FUNCTION_BLOCK JsonGraphSettingsParser IMPLEMENTS I_GraphSettings
VAR
	parser : FB_JsonDomParser;
	baseJsonValue : SJsonValue;
	jsonLanguagePack : I_JsonLanguagePack;

	_nodeCount : UDINT;
	_lastNodeId : NodeId;
	_lastLinkId : T_MAXSTRING;
	
	nodeParser : JsonNodeSettingsParser(0);
	linkParser : JsonLinkSettingsParser(0);
END_VAR

METHOD PUBLIC Clear
VAR_INPUT
END_VAR
baseJsonValue := 0;
parser.NewDocument();
END_METHOD

METHOD FB_init : BOOL
VAR_INPUT
	bInitRetains : BOOL; // if TRUE, the retain variables are initialized (warm start / cold start)
	bInCopyCode : BOOL;  // if TRUE, the instance afterwards gets moved into the copy code (online change)
	JsonLanguagePack : I_JsonLanguagePack;
END_VAR
THIS^.jsonLanguagePack := JsonLanguagePack;

nodeParser.FB_init(bInitRetains, bInCopyCode, JsonLanguagePack);
linkParser.FB_init(bInitRetains, bInCopyCode, JsonLanguagePack);
END_METHOD

METHOD PUBLIC GetLinkById : I_LinkSettings
VAR_INPUT
	Id : T_MAXSTRING;
END_VAR
VAR
	i: UDINT;
END_VAR
FOR i := 0 TO LinkCount - 1  DO
	
	linkParser.Update(parser,GetLinkObjectByIndex(i));
	
	IF linkParser.Id = Id THEN
		GetLinkById := linkParser;
		return;
	END_IF

END_FOR
END_METHOD

METHOD PUBLIC GetLinkByIndex : I_LinkSettings
VAR_INPUT
	Index : UDINT;
END_VAR
linkParser.Update(parser,GetLinkObjectByIndex(Index));
GetLinkByIndex := linkParser;
END_METHOD

METHOD PRIVATE GetLinkObjectByIndex : SJsonValue
VAR_INPUT
	Index : UDINT;
END_VAR
GetLinkObjectByIndex := parser.GetArrayValueByIdx(GetLinksArray(), Index);
END_METHOD

METHOD PRIVATE GetLinksArray : SJsonValue
GetLinksArray := parser.FindMember(baseJsonValue, 'links');
END_METHOD

METHOD PUBLIC GetNodeById : I_NodeSettings
VAR_INPUT
	Id : NodeId;
END_VAR
VAR
	i: UDINT;
END_VAR
FOR i := 0 TO NodeCount - 1  DO
	
	nodeParser.Update(parser,GetNodeObjectByIndex(i));
	
	IF nodeParser.Id = Id THEN
		GetNodeById := nodeParser;
		return;
	END_IF

END_FOR
END_METHOD

METHOD PUBLIC GetNodeByIndex : I_NodeSettings
VAR_INPUT
	Index : UDINT;
END_VAR
nodeParser.Update(parser,GetNodeObjectByIndex(Index));
GetNodeByIndex := nodeParser;
END_METHOD

METHOD PRIVATE GetNodeObjectByIndex : SJsonValue
VAR_INPUT
	Index : UDINT;
END_VAR
GetNodeObjectByIndex := parser.GetArrayValueByIdx(GetNodesArray(),Index);
END_METHOD

METHOD PRIVATE GetNodesArray : SJsonValue
GetNodesArray := parser.FindMember(baseJsonValue, 'nodes');
END_METHOD

PROPERTY PUBLIC HasLinks : Bool
GET
VAR
	tempJsonValue: SJsonValue;
END_VAR
tempJsonValue := GetLinksArray();

IF tempJsonValue = 0 OR_ELSE NOT parser.IsArray(tempJsonValue) THEN
	RETURN;	
END_IF

HasLinks := TRUE;
END_GET
END_PROPERTY

PROPERTY PUBLIC HasNodes : Bool
GET
VAR
	tempJsonValue: SJsonValue;
END_VAR
tempJsonValue := GetNodesArray();

IF tempJsonValue = 0 OR_ELSE NOT parser.IsArray(tempJsonValue) THEN
	RETURN;	
END_IF

HasNodes := TRUE;
END_GET
END_PROPERTY

PROPERTY PUBLIC LastLinkId : T_MAXSTRING
GET
VAR
	tempJsonValue: SJsonValue;
END_VAR
tempJsonValue := parser.FindMember(baseJsonValue, 'last_link_id');

IF tempJsonValue = 0 THEN
	RETURN;	
END_IF

LastLinkId := DINT_TO_STRING(parser.GetInt(tempJsonValue));
END_GET
END_PROPERTY

PROPERTY PUBLIC LastNodeId : NodeId
GET
VAR
	tempJsonValue: SJsonValue;
END_VAR
tempJsonValue := parser.FindMember(baseJsonValue, 'last_node_id');

IF tempJsonValue = 0 THEN
	RETURN;	
END_IF

LastNodeId := parser.GetInt(tempJsonValue);
END_GET
END_PROPERTY

PROPERTY PUBLIC LinkCount : UDINT
GET
IF NOT HasLinks THEN
	LinkCount := 0;
	RETURN;
END_IF

LinkCount := parser.GetArraySize(GetLinksArray());
END_GET
END_PROPERTY

METHOD PUBLIC LoadFile : BOOL;
VAR_INPUT
	FilePath : FilePath;
END_VAR
VAR
	load : BOOL := TRUE;
END_VAR
IF NOT parser.LoadDocumentFromFile(FilePath,load) THEN
	RETURN;
END_IF;

baseJsonValue := parser.GetDocumentRoot();

IF baseJsonValue <> 0 THEN
	LoadFile := TRUE;
END_IF;
END_METHOD

PROPERTY PUBLIC NodeCount : UDINT
GET
IF NOT HasNodes THEN
	NodeCount := 0;
	RETURN;
END_IF

NodeCount := parser.GetArraySize(GetNodesArray());
END_GET
END_PROPERTY

METHOD PUBLIC ReadString : BOOL
VAR_INPUT
	HugeString : REFERENCE TO HugeString;
END_VAR
baseJsonValue := parser.ParseDocument(HugeString);
ReadString := baseJsonValue <> 0;
END_METHOD

PROPERTY PUBLIC Uuid : Uuid
GET
VAR
	uuidJsonMember: SJsonValue;
END_VAR
uuidJsonMember := parser.FindMember(baseJsonValue, 'uuid');

IF uuidJsonMember = 0 THEN
	RETURN;	
END_IF

Uuid := parser.GetString(uuidJsonMember);
END_GET
END_PROPERTY

END_FUNCTION_BLOCK

(* stored: Version 1.1.0.1, ProductVersion 3.1.4024.12
   POU JsonGraphSettingsParser: Id {ebb1eb33-1a2e-0a9b-3ae0-789eca45bad7}, SpecialFunc None
   Folder Constructor: Id {06f33374-f335-0a78-1dd1-a098bddcab3a}
   Folder Private: Id {1ff1bc5a-a9a2-075f-05a5-7329c800e91d}
   Method Clear: Id {c1ed9b0c-b925-0333-1704-d0c9017e417a}
   Method FB_init: Id {dfc083b0-fcd4-0a5c-1362-5d2b13fc3723}
   Method GetLinkById: Id {543e5ed5-39e3-062d-2355-b16d06be2824}
   Method GetLinkByIndex: Id {4780680b-b1f3-0e73-218d-495f2b12f8fc}
   Method GetLinkObjectByIndex: Id {5e4ee61b-9c82-0c6c-32f4-09426b3805ff}
   Method GetLinksArray: Id {706f01ad-ef56-0f66-2330-b5d774c5a44a}
   Method GetNodeById: Id {874d8fbd-4e17-0158-0215-256af4320276}
   Method GetNodeByIndex: Id {d3e6eb7e-6604-0d50-02e1-7256ad50c802}
   Method GetNodeObjectByIndex: Id {82778c75-b362-00b8-22c9-15f9aa7c6322}
   Method GetNodesArray: Id {881e9ec4-82d4-0082-1785-8ebb6db62081}
   Property HasLinks: Id {494d8272-5b6f-0cd6-28f8-c50238936cbd}
   Get Get: Id {13ca2495-45dc-0077-031b-549dc8bf38a6}
   Property HasNodes: Id {efefb8a3-cccf-04b2-078c-c24de017ed31}
   Get Get: Id {b9873311-8e33-0920-328f-0608405d59f3}
   Property LastLinkId: Id {30ddea75-6d51-0dda-322b-eb49f99654da}
   Get Get: Id {0d2b2f69-a29b-0472-2615-9ea8c776adfe}
   Property LastNodeId: Id {7bda32bf-2419-04dc-1007-a9ae3dcf3a38}
   Get Get: Id {06fabe7e-f838-04bc-1c96-79f3bd64a7ce}
   Property LinkCount: Id {2d62cb4b-7b55-0e09-112d-fed7252a0bc8}
   Get Get: Id {eb51986e-1037-02b5-3800-deeb7fcf305e}
   Method LoadFile: Id {e6ec9504-2281-0d46-127a-1302b2bd9c84}
   Property NodeCount: Id {e00a1413-a8de-0b0e-26e6-046713363104}
   Get Get: Id {f04920bb-7f28-0702-0074-834941db56c1}
   Method ReadString: Id {b0015738-c15e-0e49-3fb7-75403a41c243}
   Property Uuid: Id {edf2eeca-e6f1-021e-1dcb-742988d10601}
   Get Get: Id {eea33af0-ae9d-0036-2e3c-9e9d5a76362c} *)
